Yaskawa INFORM job: CALIBRATE.JBI

/JOB
//NAME CALIBRATE
//POS
///NPOS 4,0,0,0,0,0
///TOOL 0
///POSTYPE PULSE
///PULSE
C00000=-45973,25480,-34069,6625,-26560,17869
C00001=-21177,96617,68300,1964,-66663,9581
C00002=21513,99872,73176,-2006,-68597,-9792
C00003=59395,7268,-46134,-7854,-27054,-23468
//INST
///DATE 2026/04/27 13:29
///ATTR SC,RW
///GROUP1 RB1
NOP
MOVJ C00000 VJ=0.78
MOVJ C00001 VJ=0.78
MOVJ C00002 VJ=0.78
MOVJ C00003 VJ=0.78
END
